Staubli VAL3: start.pgx

program start()
begin
  // Se pone en marcha la aplicacion

  // Se inicializar la aplicacion
  call inicializar()
  call ajustar()

  // Se crean las tareas de la aplicacion
  taskCreate "mcp",100,mcp()
  taskCreate "robot",100,robot()
end
